(* PLC project Beremiz Python Support Tests, beremiz Beremiz 0.0 *)
(* stored: creationDateTime 2008-12-14T16:21:19, modificationDateTime 2009-10-08T10:58:12 *)

PROGRAM main_pytest
  VAR
    python1 : python_poll;
    counter : INT;
    Block1 : python_poll;
  END_VAR
  VAR  (* added by the conversion: wires and edge detectors of the diagram *)
    _STRING_TO_INT30_ENO : BOOL;
    _STRING_TO_INT30_OUT : INT;
    _ADD32_ENO : BOOL;
    _ADD32_OUT : INT;
    _INT_TO_STRING35_ENO : BOOL;
    _INT_TO_STRING35_OUT : STRING;
    _CONCAT34_ENO : BOOL;
    _CONCAT34_OUT : STRING;
  END_VAR

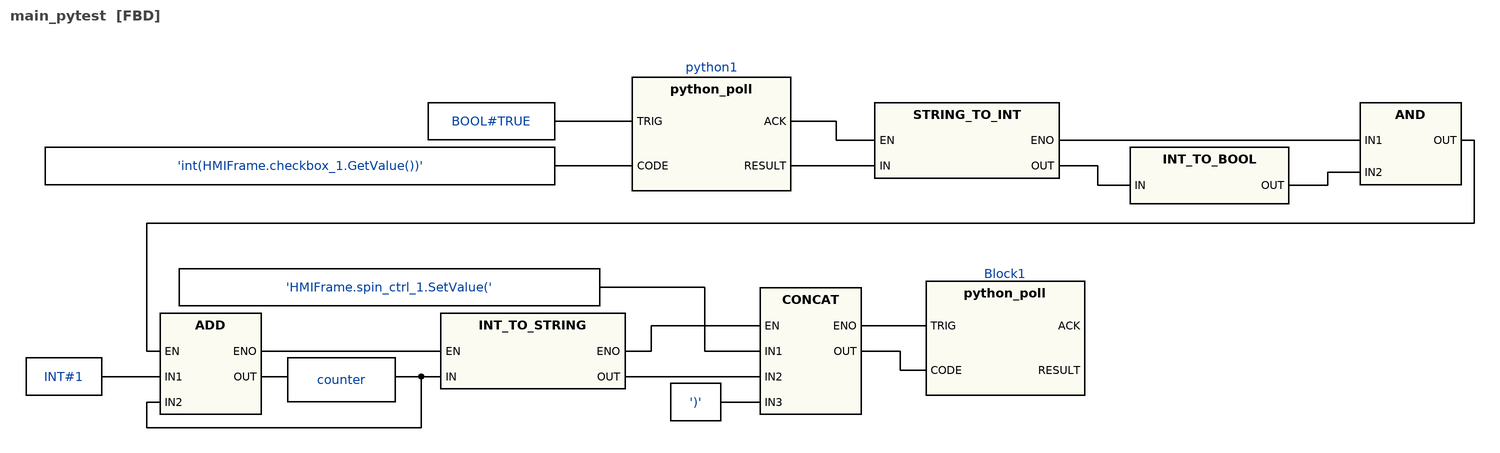
(* FBD diagram, written out as Structured Text *)
python1(TRIG := BOOL#TRUE, CODE := 'int(HMIFrame.checkbox_1.GetValue())');
_STRING_TO_INT30_OUT := STRING_TO_INT(EN := python1.ACK, IN := python1.RESULT, ENO => _STRING_TO_INT30_ENO);
_ADD32_OUT := ADD(EN := _STRING_TO_INT30_ENO AND INT_TO_BOOL(_STRING_TO_INT30_OUT), IN1 := INT#1, IN2 := counter, ENO => _ADD32_ENO);
IF _ADD32_ENO THEN counter := _ADD32_OUT; END_IF;
_INT_TO_STRING35_OUT := INT_TO_STRING(EN := _ADD32_ENO, IN := counter, ENO => _INT_TO_STRING35_ENO);
_CONCAT34_OUT := CONCAT(EN := _INT_TO_STRING35_ENO, IN1 := 'HMIFrame.spin_ctrl_1.SetValue(', IN2 := _INT_TO_STRING35_OUT, IN3 := ')', ENO => _CONCAT34_ENO);
Block1(TRIG := _CONCAT34_ENO, CODE := _CONCAT34_OUT);
END_PROGRAM

CONFIGURATION conf_pytest
  RESOURCE res_pytest ON PLC
    TASK pytest_task(INTERVAL := t#100ms, PRIORITY := 0);
    PROGRAM pytest_instance : main_pytest;
  END_RESOURCE
END_CONFIGURATION
